{attribute 'qualified_only'}
{attribute 'strict'}
TYPE E_TermType :
(
	EL320x:=0,
	EL306x:=1,
	EL305x:=2,
	EL400x:=3,
	EL401x:=4,
	EL401x_4_20:=5
);
END_TYPE

(* stored: Version 1.1.0.1, ProductVersion 3.1.4022.10
   EnumerationTextList E_TermType: Id {d5274298-b8a6-40a5-ab12-3f9f1aa3e659} *)
